# EPICS autosave request: support/ccd/1-10/ccdApp/Db/smartControl_settings_axisX.req
# FILE... smartControl_settings_axisX.req
$(P)$(R)$(AXIS)_EXISTS
$(P)$(R)$(AXIS)_OFFSET
$(P)$(R)$(AXIS)_SIGN
$(P)$(R)$(AXIS)_LOW_CUT
$(P)$(R)$(AXIS)_HIGH_CUT
